{attribute 'qualified_only'}
{attribute 'strict'}
TYPE E_ControllerMode :
(
	MANUAL,
	ACTIVE
);
END_TYPE

(* stored: Version 1.1.0.1, ProductVersion 3.1.4024.15
   DUT E_ControllerMode: Id {aa25ef5d-0bc2-0fa4-2528-5726e79c47f2} *)
